SUBAPPLICATION Uebung_004a9_AX (* mit E_SPLIT_3 *)
  (* Standard: 61499-2; Description: Copyright (c) 2026 Meisterschulen am Ostbahnhof This program and the accompanying materials are made available under the terms of the Eclipse Public License 2.0 which is available at https://www.eclipse.org/legal/epl-2.0/ SPDX-License-Identifier: EPL-2.0 *)
  (* Version 1.0, 2026-07-13, Moritz Ortmeier, Meisterschulen am Ostbahnhof *)
  PACKAGE Uebungen;
  IMPORT logiBUS::io::DI::logiBUS_DI::Input_I1;
  IMPORT logiBUS::io::DI::logiBUS_DI_Events::BUTTON_SINGLE_CLICK;
  IMPORT logiBUS::io::DQ::logiBUS_DO::Output_Q1;
  IMPORT logiBUS::io::DQ::logiBUS_DO::Output_Q2;
  IMPORT logiBUS::io::DQ::logiBUS_DO::Output_Q3;
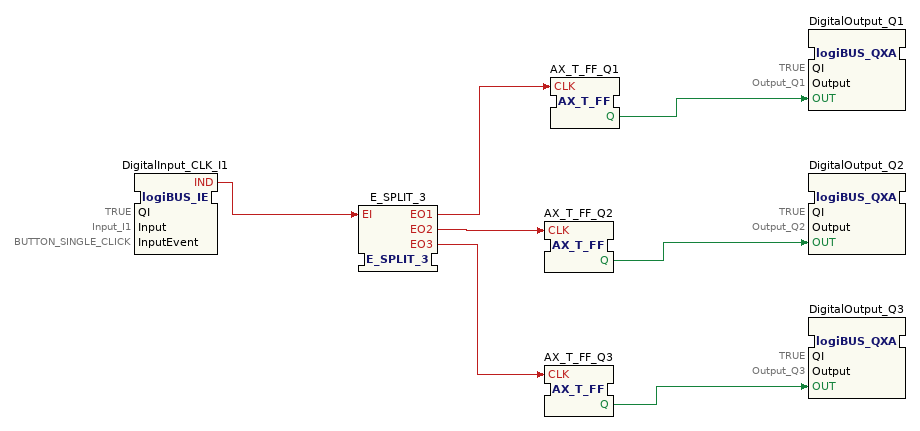
  FBS
    DigitalOutput_Q1 : logiBUS::io::DQ::logiBUS_QXA(QI := TRUE, Output := Output_Q1);
    DigitalInput_CLK_I1 : logiBUS::io::DI::logiBUS_IE(QI := TRUE, Input := Input_I1, InputEvent := BUTTON_SINGLE_CLICK);
    AX_T_FF_Q1 : adapter::events::unidirectional::AX_T_FF;
    AX_T_FF_Q2 : adapter::events::unidirectional::AX_T_FF;
    DigitalOutput_Q2 : logiBUS::io::DQ::logiBUS_QXA(QI := TRUE, Output := Output_Q2);
    AX_T_FF_Q3 : adapter::events::unidirectional::AX_T_FF;
    DigitalOutput_Q3 : logiBUS::io::DQ::logiBUS_QXA(QI := TRUE, Output := Output_Q3);
    E_SPLIT_3 : iec61499::events::E_SPLIT_3;
  END_FBS
  EVENT_CONNECTIONS
    DigitalInput_CLK_I1.IND TO E_SPLIT_3.EI;
    E_SPLIT_3.EO1 TO AX_T_FF_Q1.CLK;
    E_SPLIT_3.EO2 TO AX_T_FF_Q2.CLK;
    E_SPLIT_3.EO3 TO AX_T_FF_Q3.CLK;
  END_CONNECTIONS
  ADAPTER_CONNECTIONS
    AX_T_FF_Q3.Q TO DigitalOutput_Q3.OUT;
    AX_T_FF_Q2.Q TO DigitalOutput_Q2.OUT;
    AX_T_FF_Q1.Q TO DigitalOutput_Q1.OUT;
  END_CONNECTIONS
END_SUBAPPLICATION
